//Place your alarm trigger logic here. 
IF io_mapping.pt_3414_b.scaled_value >= opc.popa_0092_pt_3414_b_high_high_setpoint THEN
    pt_3414_b_high_high.trigger := TRUE;
    ELSE
        pt_3414_b_high_high.trigger := FALSE;
END_IF

(*

//pt_3428-----------------------------------------------------------------------------------------------------
//Instantiate the alarm block, and map the inputs from the OPC GVL
pt_3428_b_low_low();
pt_3428_b_low_low.alm_ack:=opc.popa_0082_alarm_ack;
pt_3428_b_low_low.reset:=opc.popa_0082_alarm_reset;
pt_3428_b_low_low.priority:=opc.popa_0082_pt_3428_b_low_low_priority;
pt_3428_b_low_low.delay_setpoint:=opc.popa_0082_pt_3428_b_low_low_setpoint;
pt_3428_b_low_low.enable:=opc.popa_0082_pt_3428_b_low_low_enable;

//Timer delay elapsed
pt_3428_b_low_low.delay_ton_et;

//Place your alarm trigger logic here. 
IF io_mapping.pt_3428.scaled_value <= opc.popa_0082_pt_3428_b_low_low_setpoint THEN
    pt_3428_b_low_low.trigger := TRUE;
    ELSE
        pt_3428_b_low_low.trigger := FALSE;
END_IF
	
//pt_3428-----------------------------------------------------------------------------------------------------
//Instantiate the alarm block, and map the inputs from the OPC GVL
pt_3428_b_low();
pt_3428_b_low.alm_ack:=opc.popa_0082_alarm_ack;
pt_3428_b_low.reset:=opc.popa_0082_alarm_reset;
pt_3428_b_low.priority:=opc.popa_0082_pt_3428_b_low_priority;
pt_3428_b_low.delay_setpoint:=opc.popa_0082_pt_3428_b_low_setpoint;
pt_3428_b_low.enable:=opc.popa_0082_pt_3428_b_low_enable;

//Timer delay elapsed
pt_3428_b_low.delay_ton_et;

//Place your alarm trigger logic here. 
IF io_mapping.pt_3428.scaled_value < opc.popa_0082_pt_3428_b_low_setpoint THEN
    pt_3428_b_low.trigger := TRUE;
    ELSE
        pt_3428_b_low.trigger := FALSE;
END_IF
	
//pt_3428-----------------------------------------------------------------------------------------------------
//Instantiate the alarm block, and map the inputs from the OPC GVL
pt_3428_b_high();
pt_3428_b_high.alm_ack:=opc.popa_0082_alarm_ack;
pt_3428_b_high.reset:=opc.popa_0082_alarm_reset;
pt_3428_b_high.priority:=opc.popa_0082_pt_3428_b_high_priority;
pt_3428_b_high.delay_setpoint:=opc.popa_0082_pt_3428_b_high_setpoint;
pt_3428_b_high.enable:=opc.popa_0082_pt_3428_b_high_enable;

//Timer delay elapsed
pt_3428_b_high.delay_ton_et;

//Place your alarm trigger logic here. 
IF io_mapping.pt_3428.scaled_value > opc.popa_0082_pt_3428_b_high_setpoint THEN
    pt_3428_b_high.trigger := TRUE;
    ELSE
        pt_3428_b_high.trigger := FALSE;
END_IF
	
//pt_3428-----------------------------------------------------------------------------------------------------
//Instantiate the alarm block, and map the inputs from the OPC GVL
pt_3428_b_high_high();
pt_3428_b_high_high.alm_ack:=opc.popa_0082_alarm_ack;
pt_3428_b_high_high.reset:=opc.popa_0082_alarm_reset;
pt_3428_b_high_high.priority:=opc.popa_0082_pt_3428_b_high_high_priority;
pt_3428_b_high_high.delay_setpoint:=opc.popa_0082_pt_3428_b_high_high_setpoint;
pt_3428_b_high_high.enable:=opc.popa_0082_pt_3428_b_high_high_enable;

//Timer delay elapsed
pt_3428_b_high_high.delay_ton_et;

//Place your alarm trigger logic here. 
IF io_mapping.pt_3428.scaled_value >= opc.popa_0082_pt_3428_b_high_high_setpoint THEN
    pt_3428_b_high_high.trigger := TRUE;
    ELSE
        pt_3428_b_high_high.trigger := FALSE;
END_IF

*)
//tt_3118-----------------------------------------------------------------------------------------------------
//Instantiate the alarm block, and map the inputs from the OPC GVL
tt_3118_b_low_low();
tt_3118_b_low_low.alm_ack:=opc.popa_0082_alarm_ack;
tt_3118_b_low_low.reset:=opc.popa_0082_alarm_reset;
tt_3118_b_low_low.priority:=opc.popa_0082_tt_3118_b_low_low_priority;
tt_3118_b_low_low.delay_setpoint:=opc.popa_0082_tt_3118_b_low_low_setpoint;
tt_3118_b_low_low.enable:=opc.popa_0082_tt_3118_b_low_low_enable;

//Timer delay elapsed
tt_3118_b_low_low.delay_ton_et;

//Place your alarm trigger logic here. 
IF io_mapping.tt_3118_b.scaled_value <= opc.popa_0082_tt_3118_b_low_low_setpoint THEN
    tt_3118_b_low_low.trigger := TRUE;
    ELSE
        tt_3118_b_low_low.trigger := FALSE;
END_IF
	
//tt_3118-----------------------------------------------------------------------------------------------------
//Instantiate the alarm block, and map the inputs from the OPC GVL
tt_3118_b_low();
tt_3118_b_low.alm_ack:=opc.popa_0082_alarm_ack;
tt_3118_b_low.reset:=opc.popa_0082_alarm_reset;
tt_3118_b_low.priority:=opc.popa_0082_tt_3118_b_low_priority;
tt_3118_b_low.delay_setpoint:=opc.popa_0082_tt_3118_b_low_setpoint;
tt_3118_b_low.enable:=opc.popa_0082_tt_3118_b_low_enable;

//Timer delay elapsed
tt_3118_b_low.delay_ton_et;

//Place your alarm trigger logic here. 
IF io_mapping.tt_3118_b.scaled_value < opc.popa_0082_tt_3118_b_low_setpoint THEN
    tt_3118_b_low.trigger := TRUE;
    ELSE
        tt_3118_b_low.trigger := FALSE;
END_IF
	
//tt_3118-----------------------------------------------------------------------------------------------------
//Instantiate the alarm block, and map the inputs from the OPC GVL
tt_3118_b_high();
tt_3118_b_high.alm_ack:=opc.popa_0082_alarm_ack;
tt_3118_b_high.reset:=opc.popa_0082_alarm_reset;
tt_3118_b_high.priority:=opc.popa_0082_tt_3118_b_high_priority;
tt_3118_b_high.delay_setpoint:=opc.popa_0082_tt_3118_b_high_setpoint;
tt_3118_b_high.enable:=opc.popa_0082_tt_3118_b_high_enable;

//Timer delay elapsed
tt_3118_b_high.delay_ton_et;

//Place your alarm trigger logic here. 
IF io_mapping.tt_3118_b.scaled_value > opc.popa_0082_tt_3118_b_high_setpoint THEN
    tt_3118_b_high.trigger := TRUE;
    ELSE
        tt_3118_b_high.trigger := FALSE;
END_IF
	
//tt_3118-----------------------------------------------------------------------------------------------------
//Instantiate the alarm block, and map the inputs from the OPC GVL
tt_3118_b_high_high();
tt_3118_b_high_high.alm_ack:=opc.popa_0082_alarm_ack;
tt_3118_b_high_high.reset:=opc.popa_0082_alarm_reset;
tt_3118_b_high_high.priority:=opc.popa_0082_tt_3118_b_high_high_priority;
tt_3118_b_high_high.delay_setpoint:=opc.popa_0082_tt_3118_b_high_high_setpoint;
tt_3118_b_high_high.enable:=opc.popa_0082_tt_3118_b_high_high_enable;

//Timer delay elapsed
tt_3118_b_high_high.delay_ton_et;

//Place your alarm trigger logic here. 
IF io_mapping.tt_3118_b.scaled_value >= opc.popa_0082_tt_3118_b_high_high_setpoint THEN
    tt_3118_b_high_high.trigger := TRUE;
    ELSE
        tt_3118_b_high_high.trigger := FALSE;
END_IF


//tt_3218-----------------------------------------------------------------------------------------------------
//Instantiate the alarm block, and map the inputs from the OPC GVL
tt_3218_b_low_low();
tt_3218_b_low_low.alm_ack:=opc.popa_0082_alarm_ack;
tt_3218_b_low_low.reset:=opc.popa_0082_alarm_reset;
tt_3218_b_low_low.priority:=opc.popa_0082_tt_3218_b_low_low_priority;
tt_3218_b_low_low.delay_setpoint:=opc.popa_0082_tt_3218_b_low_low_setpoint;
tt_3218_b_low_low.enable:=opc.popa_0082_tt_3218_b_low_low_enable;

//Timer delay elapsed
tt_3218_b_low_low.delay_ton_et;

//Place your alarm trigger logic here. 
IF io_mapping.tt_3218_b.scaled_value <= opc.popa_0082_tt_3218_b_low_low_setpoint THEN
    tt_3218_b_low_low.trigger := TRUE;
    ELSE
        tt_3218_b_low_low.trigger := FALSE;
END_IF
	
//tt_3218-----------------------------------------------------------------------------------------------------
//Instantiate the alarm block, and map the inputs from the OPC GVL
tt_3218_b_low();
tt_3218_b_low.alm_ack:=opc.popa_0082_alarm_ack;
tt_3218_b_low.reset:=opc.popa_0082_alarm_reset;
tt_3218_b_low.priority:=opc.popa_0082_tt_3218_b_low_priority;
tt_3218_b_low.delay_setpoint:=opc.popa_0082_tt_3218_b_low_setpoint;
tt_3218_b_low.enable:=opc.popa_0082_tt_3218_b_low_enable;

//Timer delay elapsed
tt_3218_b_low.delay_ton_et;

//Place your alarm trigger logic here. 
IF io_mapping.tt_3218_b.scaled_value < opc.popa_0082_tt_3218_b_low_setpoint THEN
    tt_3218_b_low.trigger := TRUE;
    ELSE
        tt_3218_b_low.trigger := FALSE;
END_IF
	
//tt_3218-----------------------------------------------------------------------------------------------------
//Instantiate the alarm block, and map the inputs from the OPC GVL
tt_3218_b_high();
tt_3218_b_high.alm_ack:=opc.popa_0082_alarm_ack;
tt_3218_b_high.reset:=opc.popa_0082_alarm_reset;
tt_3218_b_high.priority:=opc.popa_0082_tt_3218_b_high_priority;
tt_3218_b_high.delay_setpoint:=opc.popa_0082_tt_3218_b_high_setpoint;
tt_3218_b_high.enable:=opc.popa_0082_tt_3218_b_high_enable;

//Timer delay elapsed
tt_3218_b_high.delay_ton_et;

//Place your alarm trigger logic here. 
IF io_mapping.tt_3218_b.scaled_value > opc.popa_0082_tt_3218_b_high_setpoint THEN
    tt_3218_b_high.trigger := TRUE;
    ELSE
        tt_3218_b_high.trigger := FALSE;
END_IF
	
//tt_3218-----------------------------------------------------------------------------------------------------
//Instantiate the alarm block, and map the inputs from the OPC GVL
tt_3218_b_high_high();
tt_3218_b_high_high.alm_ack:=opc.popa_0082_alarm_ack;
tt_3218_b_high_high.reset:=opc.popa_0082_alarm_reset;
tt_3218_b_high_high.priority:=opc.popa_0082_tt_3218_b_high_high_priority;
tt_3218_b_high_high.delay_setpoint:=opc.popa_0082_tt_3218_b_high_high_setpoint;
tt_3218_b_high_high.enable:=opc.popa_0082_tt_3218_b_high_high_enable;

//Timer delay elapsed
tt_3218_b_high_high.delay_ton_et;

//Place your alarm trigger logic here. 
IF io_mapping.tt_3218_b.scaled_value >= opc.popa_0082_tt_3218_b_high_high_setpoint THEN
    tt_3218_b_high_high.trigger := TRUE;
    ELSE
        tt_3218_b_high_high.trigger := FALSE;
END_IF


//tt_3318-----------------------------------------------------------------------------------------------------
//Instantiate the alarm block, and map the inputs from the OPC GVL
tt_3318_b_low_low();
tt_3318_b_low_low.alm_ack:=opc.popa_0082_alarm_ack;
tt_3318_b_low_low.reset:=opc.popa_0082_alarm_reset;
tt_3318_b_low_low.priority:=opc.popa_0082_tt_3318_b_low_low_priority;
tt_3318_b_low_low.delay_setpoint:=opc.popa_0082_tt_3318_b_low_low_setpoint;
tt_3318_b_low_low.enable:=opc.popa_0082_tt_3318_b_low_low_enable;

//Timer delay elapsed
tt_3318_b_low_low.delay_ton_et;

//Place your alarm trigger logic here. 
IF io_mapping.tt_3318_b.scaled_value <= opc.popa_0082_tt_3318_b_low_low_setpoint THEN
    tt_3318_b_low_low.trigger := TRUE;
    ELSE
        tt_3318_b_low_low.trigger := FALSE;
END_IF
	
//tt_3318-----------------------------------------------------------------------------------------------------
//Instantiate the alarm block, and map the inputs from the OPC GVL
tt_3318_b_low();
tt_3318_b_low.alm_ack:=opc.popa_0082_alarm_ack;
tt_3318_b_low.reset:=opc.popa_0082_alarm_reset;
tt_3318_b_low.priority:=opc.popa_0082_tt_3318_b_low_priority;
tt_3318_b_low.delay_setpoint:=opc.popa_0082_tt_3318_b_low_setpoint;
tt_3318_b_low.enable:=opc.popa_0082_tt_3318_b_low_enable;

//Timer delay elapsed
tt_3318_b_low.delay_ton_et;

//Place your alarm trigger logic here. 
IF io_mapping.tt_3318_b.scaled_value < opc.popa_0082_tt_3318_b_low_setpoint THEN
    tt_3318_b_low.trigger := TRUE;
    ELSE
        tt_3318_b_low.trigger := FALSE;
END_IF
	
//tt_3318-----------------------------------------------------------------------------------------------------
//Instantiate the alarm block, and map the inputs from the OPC GVL
tt_3318_b_high();
tt_3318_b_high.alm_ack:=opc.popa_0082_alarm_ack;
tt_3318_b_high.reset:=opc.popa_0082_alarm_reset;
tt_3318_b_high.priority:=opc.popa_0082_tt_3318_b_high_priority;
tt_3318_b_high.delay_setpoint:=opc.popa_0082_tt_3318_b_high_setpoint;
tt_3318_b_high.enable:=opc.popa_0082_tt_3318_b_high_enable;

//Timer delay elapsed
tt_3318_b_high.delay_ton_et;

//Place your alarm trigger logic here. 
IF io_mapping.tt_3318_b.scaled_value > opc.popa_0082_tt_3318_b_high_setpoint THEN
    tt_3318_b_high.trigger := TRUE;
    ELSE
        tt_3318_b_high.trigger := FALSE;
END_IF
	
//tt_3318-----------------------------------------------------------------------------------------------------
//Instantiate the alarm block, and map the inputs from the OPC GVL
tt_3318_b_high_high();
tt_3318_b_high_high.alm_ack:=opc.popa_0082_alarm_ack;
tt_3318_b_high_high.reset:=opc.popa_0082_alarm_reset;
tt_3318_b_high_high.priority:=opc.popa_0082_tt_3318_b_high_high_priority;
tt_3318_b_high_high.delay_setpoint:=opc.popa_0082_tt_3318_b_high_high_setpoint;
tt_3318_b_high_high.enable:=opc.popa_0082_tt_3318_b_high_high_enable;

//Timer delay elapsed
tt_3318_b_high_high.delay_ton_et;

//Place your alarm trigger logic here. 
IF io_mapping.tt_3318_b.scaled_value >= opc.popa_0082_tt_3318_b_high_high_setpoint THEN
    tt_3318_b_high_high.trigger := TRUE;
    ELSE
        tt_3318_b_high_high.trigger := FALSE;
END_IF


//tt_3140-----------------------------------------------------------------------------------------------------
//Instantiate the alarm block, and map the inputs from the OPC GVL
tt_3140_b_low_low();
tt_3140_b_low_low.alm_ack:=opc.popa_0082_alarm_ack;
tt_3140_b_low_low.reset:=opc.popa_0082_alarm_reset;
tt_3140_b_low_low.priority:=opc.popa_0082_tt_3140_b_low_low_priority;
tt_3140_b_low_low.delay_setpoint:=opc.popa_0082_tt_3140_b_low_low_setpoint;
tt_3140_b_low_low.enable:=opc.popa_0082_tt_3140_b_low_low_enable;

//Timer delay elapsed
tt_3140_b_low_low.delay_ton_et;

//Place your alarm trigger logic here. 
IF io_mapping.tt_3140_b.scaled_value <= opc.popa_0082_tt_3140_b_low_low_setpoint THEN
    tt_3140_b_low_low.trigger := TRUE;
    ELSE
        tt_3140_b_low_low.trigger := FALSE;
END_IF
	
//tt_3140-----------------------------------------------------------------------------------------------------
//Instantiate the alarm block, and map the inputs from the OPC GVL
tt_3140_b_low();
tt_3140_b_low.alm_ack:=opc.popa_0082_alarm_ack;
tt_3140_b_low.reset:=opc.popa_0082_alarm_reset;
tt_3140_b_low.priority:=opc.popa_0082_tt_3140_b_low_priority;
tt_3140_b_low.delay_setpoint:=opc.popa_0082_tt_3140_b_low_setpoint;
tt_3140_b_low.enable:=opc.popa_0082_tt_3140_b_low_enable;

//Timer delay elapsed
tt_3140_b_low.delay_ton_et;

//Place your alarm trigger logic here. 
IF io_mapping.tt_3140_b.scaled_value < opc.popa_0082_tt_3140_b_low_setpoint THEN
    tt_3140_b_low.trigger := TRUE;
    ELSE
        tt_3140_b_low.trigger := FALSE;
END_IF
	
//tt_3140-----------------------------------------------------------------------------------------------------
//Instantiate the alarm block, and map the inputs from the OPC GVL
tt_3140_b_high();
tt_3140_b_high.alm_ack:=opc.popa_0082_alarm_ack;
tt_3140_b_high.reset:=opc.popa_0082_alarm_reset;
tt_3140_b_high.priority:=opc.popa_0082_tt_3140_b_high_priority;
tt_3140_b_high.delay_setpoint:=opc.popa_0082_tt_3140_b_high_setpoint;
tt_3140_b_high.enable:=opc.popa_0082_tt_3140_b_high_enable;

//Timer delay elapsed
tt_3140_b_high.delay_ton_et;

//Place your alarm trigger logic here. 
IF io_mapping.tt_3140_b.scaled_value > opc.popa_0082_tt_3140_b_high_setpoint THEN
    tt_3140_b_high.trigger := TRUE;
    ELSE
        tt_3140_b_high.trigger := FALSE;
END_IF
	
//tt_3140-----------------------------------------------------------------------------------------------------
//Instantiate the alarm block, and map the inputs from the OPC GVL
tt_3140_b_high_high();
tt_3140_b_high_high.alm_ack:=opc.popa_0082_alarm_ack;
tt_3140_b_high_high.reset:=opc.popa_0082_alarm_reset;
tt_3140_b_high_high.priority:=opc.popa_0082_tt_3140_b_high_high_priority;
tt_3140_b_high_high.delay_setpoint:=opc.popa_0082_tt_3140_b_high_high_setpoint;
tt_3140_b_high_high.enable:=opc.popa_0082_tt_3140_b_high_high_enable;

//Timer delay elapsed
tt_3140_b_high_high.delay_ton_et;

//Place your alarm trigger logic here. 
IF io_mapping.tt_3140_b.scaled_value >= opc.popa_0082_tt_3140_b_high_high_setpoint THEN
    tt_3140_b_high_high.trigger := TRUE;
    ELSE
        tt_3140_b_high_high.trigger := FALSE;
END_IF


//tt_3240-----------------------------------------------------------------------------------------------------
//Instantiate the alarm block, and map the inputs from the OPC GVL
tt_3240_b_low_low();
tt_3240_b_low_low.alm_ack:=opc.popa_0082_alarm_ack;
tt_3240_b_low_low.reset:=opc.popa_0082_alarm_reset;
tt_3240_b_low_low.priority:=opc.popa_0082_tt_3240_b_low_low_priority;
tt_3240_b_low_low.delay_setpoint:=opc.popa_0082_tt_3240_b_low_low_setpoint;
tt_3240_b_low_low.enable:=opc.popa_0082_tt_3240_b_low_low_enable;

//Timer delay elapsed
tt_3240_b_low_low.delay_ton_et;

//Place your alarm trigger logic here. 
IF io_mapping.tt_3240_b.scaled_value <= opc.popa_0082_tt_3240_b_low_low_setpoint THEN
    tt_3240_b_low_low.trigger := TRUE;
    ELSE
        tt_3240_b_low_low.trigger := FALSE;
END_IF
	
//tt_3240-----------------------------------------------------------------------------------------------------
//Instantiate the alarm block, and map the inputs from the OPC GVL
tt_3240_b_low();
tt_3240_b_low.alm_ack:=opc.popa_0082_alarm_ack;
tt_3240_b_low.reset:=opc.popa_0082_alarm_reset;
tt_3240_b_low.priority:=opc.popa_0082_tt_3240_b_low_priority;
tt_3240_b_low.delay_setpoint:=opc.popa_0082_tt_3240_b_low_setpoint;
tt_3240_b_low.enable:=opc.popa_0082_tt_3240_b_low_enable;

//Timer delay elapsed
tt_3240_b_low.delay_ton_et;

//Place your alarm trigger logic here. 
IF io_mapping.tt_3240_b.scaled_value < opc.popa_0082_tt_3240_b_low_setpoint THEN
    tt_3240_b_low.trigger := TRUE;
    ELSE
        tt_3240_b_low.trigger := FALSE;
END_IF
	
//tt_3240-----------------------------------------------------------------------------------------------------
//Instantiate the alarm block, and map the inputs from the OPC GVL
tt_3240_b_high();
tt_3240_b_high.alm_ack:=opc.popa_0082_alarm_ack;
tt_3240_b_high.reset:=opc.popa_0082_alarm_reset;
tt_3240_b_high.priority:=opc.popa_0082_tt_3240_b_high_priority;
tt_3240_b_high.delay_setpoint:=opc.popa_0082_tt_3240_b_high_setpoint;
tt_3240_b_high.enable:=opc.popa_0082_tt_3240_b_high_enable;

//Timer delay elapsed
tt_3240_b_high.delay_ton_et;

//Place your alarm trigger logic here. 
IF io_mapping.tt_3240_b.scaled_value > opc.popa_0082_tt_3240_b_high_setpoint THEN
    tt_3240_b_high.trigger := TRUE;
    ELSE
        tt_3240_b_high.trigger := FALSE;
END_IF
	
//tt_3240-----------------------------------------------------------------------------------------------------
//Instantiate the alarm block, and map the inputs from the OPC GVL
tt_3240_b_high_high();
tt_3240_b_high_high.alm_ack:=opc.popa_0082_alarm_ack;
tt_3240_b_high_high.reset:=opc.popa_0082_alarm_reset;
tt_3240_b_high_high.priority:=opc.popa_0082_tt_3240_b_high_high_priority;
tt_3240_b_high_high.delay_setpoint:=opc.popa_0082_tt_3240_b_high_high_setpoint;
tt_3240_b_high_high.enable:=opc.popa_0082_tt_3240_b_high_high_enable;

//Timer delay elapsed
tt_3240_b_high_high.delay_ton_et;

//Place your alarm trigger logic here. 
IF io_mapping.tt_3240_b.scaled_value >= opc.popa_0082_tt_3240_b_high_high_setpoint THEN
    tt_3240_b_high_high.trigger := TRUE;
    ELSE
        tt_3240_b_high_high.trigger := FALSE;
END_IF


//tt_3340-----------------------------------------------------------------------------------------------------
//Instantiate the alarm block, and map the inputs from the OPC GVL
tt_3340_b_low_low();
tt_3340_b_low_low.alm_ack:=opc.popa_0082_alarm_ack;
tt_3340_b_low_low.reset:=opc.popa_0082_alarm_reset;
tt_3340_b_low_low.priority:=opc.popa_0082_tt_3340_b_low_low_priority;
tt_3340_b_low_low.delay_setpoint:=opc.popa_0082_tt_3340_b_low_low_setpoint;
tt_3340_b_low_low.enable:=opc.popa_0082_tt_3340_b_low_low_enable;

//Timer delay elapsed
tt_3340_b_low_low.delay_ton_et;

//Place your alarm trigger logic here. 
IF io_mapping.tt_3340_b.scaled_value <= opc.popa_0082_tt_3340_b_low_low_setpoint THEN
    tt_3340_b_low_low.trigger := TRUE;
    ELSE
        tt_3340_b_low_low.trigger := FALSE;
END_IF
	
//tt_3340-----------------------------------------------------------------------------------------------------
//Instantiate the alarm block, and map the inputs from the OPC GVL
tt_3340_b_low();
tt_3340_b_low.alm_ack:=opc.popa_0082_alarm_ack;
tt_3340_b_low.reset:=opc.popa_0082_alarm_reset;
tt_3340_b_low.priority:=opc.popa_0082_tt_3340_b_low_priority;
tt_3340_b_low.delay_setpoint:=opc.popa_0082_tt_3340_b_low_setpoint;
tt_3340_b_low.enable:=opc.popa_0082_tt_3340_b_low_enable;

//Timer delay elapsed
tt_3340_b_low.delay_ton_et;

//Place your alarm trigger logic here. 
IF io_mapping.tt_3340_b.scaled_value < opc.popa_0082_tt_3340_b_low_setpoint THEN
    tt_3340_b_low.trigger := TRUE;
    ELSE
        tt_3340_b_low.trigger := FALSE;
END_IF
	
//tt_3340-----------------------------------------------------------------------------------------------------
//Instantiate the alarm block, and map the inputs from the OPC GVL
tt_3340_b_high();
tt_3340_b_high.alm_ack:=opc.popa_0082_alarm_ack;
tt_3340_b_high.reset:=opc.popa_0082_alarm_reset;
tt_3340_b_high.priority:=opc.popa_0082_tt_3340_b_high_priority;
tt_3340_b_high.delay_setpoint:=opc.popa_0082_tt_3340_b_high_setpoint;
tt_3340_b_high.enable:=opc.popa_0082_tt_3340_b_high_enable;

//Timer delay elapsed
tt_3340_b_high.delay_ton_et;

//Place your alarm trigger logic here. 
IF io_mapping.tt_3340_b.scaled_value > opc.popa_0082_tt_3340_b_high_setpoint THEN
    tt_3340_b_high.trigger := TRUE;
    ELSE
        tt_3340_b_high.trigger := FALSE;
END_IF
	
//tt_3340-----------------------------------------------------------------------------------------------------
//Instantiate the alarm block, and map the inputs from the OPC GVL
tt_3340_b_high_high();
tt_3340_b_high_high.alm_ack:=opc.popa_0082_alarm_ack;
tt_3340_b_high_high.reset:=opc.popa_0082_alarm_reset;
tt_3340_b_high_high.priority:=opc.popa_0082_tt_3340_b_high_high_priority;
tt_3340_b_high_high.delay_setpoint:=opc.popa_0082_tt_3340_b_high_high_setpoint;
tt_3340_b_high_high.enable:=opc.popa_0082_tt_3340_b_high_high_enable;

//Timer delay elapsed
tt_3340_b_high_high.delay_ton_et;

//Place your alarm trigger logic here. 
IF io_mapping.tt_3340_b.scaled_value >= opc.popa_0082_tt_3340_b_high_high_setpoint THEN
    tt_3340_b_high_high.trigger := TRUE;
    ELSE
        tt_3340_b_high_high.trigger := FALSE;
END_IF


//tt_3432-----------------------------------------------------------------------------------------------------
//Instantiate the alarm block, and map the inputs from the OPC GVL
tt_3432_b_low_low();
tt_3432_b_low_low.alm_ack:=opc.popa_0082_alarm_ack;
tt_3432_b_low_low.reset:=opc.popa_0082_alarm_reset;
tt_3432_b_low_low.priority:=opc.popa_0092_tt_3432_b_low_low_priority;
tt_3432_b_low_low.delay_setpoint:=opc.popa_0092_tt_3432_b_low_low_setpoint;
tt_3432_b_low_low.enable:=opc.popa_0092_tt_3432_b_low_low_enable;

//Timer delay elapsed
tt_3432_b_low_low.delay_ton_et;

//Place your alarm trigger logic here. 
IF io_mapping.tt_3432_b.scaled_value <= opc.popa_0092_tt_3432_b_low_low_setpoint THEN
    tt_3432_b_low_low.trigger := TRUE;
    ELSE
        tt_3432_b_low_low.trigger := FALSE;
END_IF
	
//tt_3432-----------------------------------------------------------------------------------------------------
//Instantiate the alarm block, and map the inputs from the OPC GVL
tt_3432_b_low();
tt_3432_b_low.alm_ack:=opc.popa_0082_alarm_ack;
tt_3432_b_low.reset:=opc.popa_0082_alarm_reset;
tt_3432_b_low.priority:=opc.popa_0092_tt_3432_b_low_priority;
tt_3432_b_low.delay_setpoint:=opc.popa_0092_tt_3432_b_low_setpoint;
tt_3432_b_low.enable:=opc.popa_0092_tt_3432_b_low_enable;

//Timer delay elapsed
tt_3432_b_low.delay_ton_et;

//Place your alarm trigger logic here. 
IF io_mapping.tt_3432_b.scaled_value < opc.popa_0092_tt_3432_b_low_setpoint THEN
    tt_3432_b_low.trigger := TRUE;
    ELSE
        tt_3432_b_low.trigger := FALSE;
END_IF
	
//tt_3432-----------------------------------------------------------------------------------------------------
//Instantiate the alarm block, and map the inputs from the OPC GVL
tt_3432_b_high();
tt_3432_b_high.alm_ack:=opc.popa_0082_alarm_ack;
tt_3432_b_high.reset:=opc.popa_0082_alarm_reset;
tt_3432_b_high.priority:=opc.popa_0092_tt_3432_b_high_priority;
tt_3432_b_high.delay_setpoint:=opc.popa_0092_tt_3432_b_high_setpoint;
tt_3432_b_high.enable:=opc.popa_0092_tt_3432_b_high_enable;

//Timer delay elapsed
tt_3432_b_high.delay_ton_et;

//Place your alarm trigger logic here. 
IF io_mapping.tt_3432_b.scaled_value > opc.popa_0092_tt_3432_b_high_setpoint THEN
    tt_3432_b_high.trigger := TRUE;
    ELSE
        tt_3432_b_high.trigger := FALSE;
END_IF
	
//tt_3432-----------------------------------------------------------------------------------------------------
//Instantiate the alarm block, and map the inputs from the OPC GVL
tt_3432_b_high_high();
tt_3432_b_high_high.alm_ack:=opc.popa_0082_alarm_ack;
tt_3432_b_high_high.reset:=opc.popa_0082_alarm_reset;
tt_3432_b_high_high.priority:=opc.popa_0092_tt_3432_b_high_high_priority;
tt_3432_b_high_high.delay_setpoint:=opc.popa_0092_tt_3432_b_high_high_setpoint;
tt_3432_b_high_high.enable:=opc.popa_0092_tt_3432_b_high_high_enable;

//Timer delay elapsed
tt_3432_b_high_high.delay_ton_et;

//Place your alarm trigger logic here. 
IF io_mapping.tt_3432_b.scaled_value >= opc.popa_0092_tt_3432_b_high_high_setpoint THEN
    tt_3432_b_high_high.trigger := TRUE;
    ELSE
        tt_3432_b_high_high.trigger := FALSE;
END_IF

END_PROGRAM

(* stored: Version 1.1.0.1, ProductVersion 3.1.4024.15
   POU faults: Id {676b0c44-de53-481b-87a6-7f945cc11bcf}, SpecialFunc None *)
